// Mitsubishi GX Works2 project: pneumatic_control_3   PLC: Q03UDV

PROGRAM MAIN
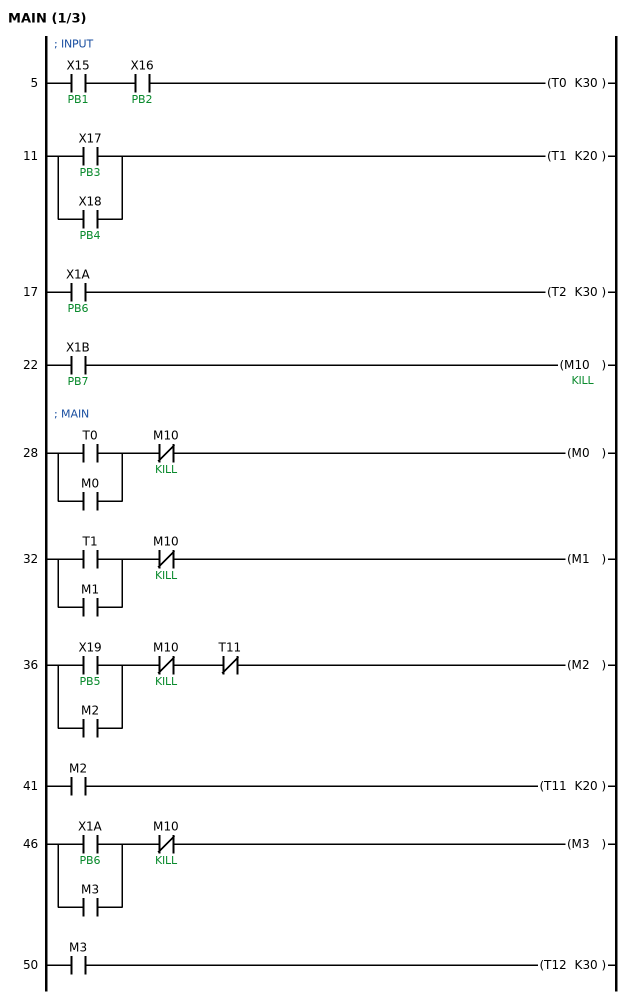
; INPUT
5     LD      X15  ; PB1
      AND     X16  ; PB2
      OUT     T0 K30
11    LD      X17  ; PB3
      OR      X18  ; PB4
      OUT     T1 K20
17    LD      X1A  ; PB6
      OUT     T2 K30
22    LD      X1B  ; PB7
      OUT     M10  ; KILL
; MAIN
28    LD      T0
      OR      M0
      ANI     M10  ; KILL
      OUT     M0
32    LD      T1
      OR      M1
      ANI     M10  ; KILL
      OUT     M1
36    LD      X19  ; PB5
      OR      M2
      ANI     M10  ; KILL
      ANI     T11
      OUT     M2
41    LD      M2
      OUT     T11 K20
46    LD      X1A  ; PB6
      OR      M3
      ANI     M10  ; KILL
      OUT     M3
50    LD      M3
      OUT     T12 K30
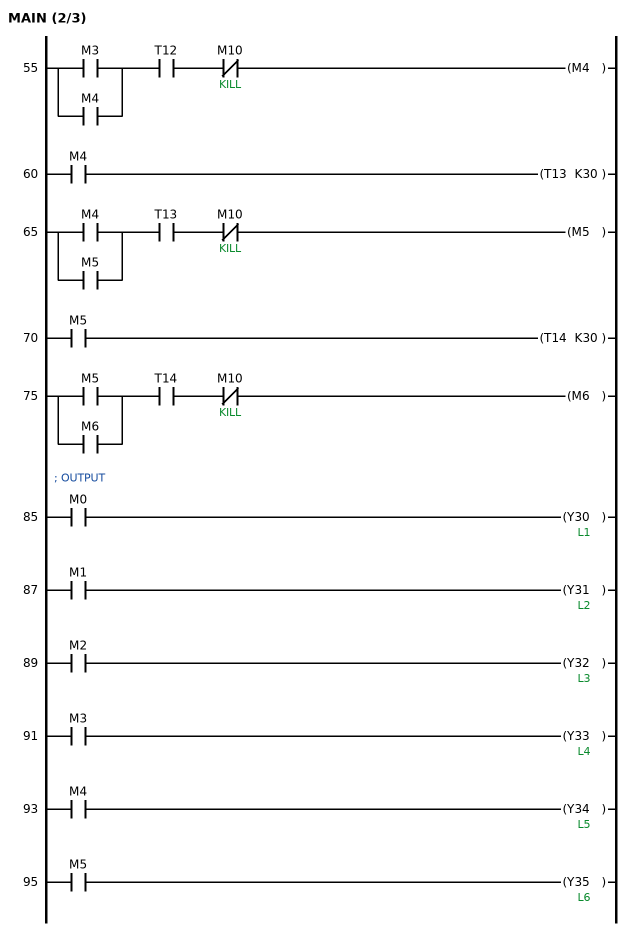
55    LD      M3
      OR      M4
      AND     T12
      ANI     M10  ; KILL
      OUT     M4
60    LD      M4
      OUT     T13 K30
65    LD      M4
      OR      M5
      AND     T13
      ANI     M10  ; KILL
      OUT     M5
70    LD      M5
      OUT     T14 K30
75    LD      M5
      OR      M6
      AND     T14
      ANI     M10  ; KILL
      OUT     M6
; OUTPUT
85    LD      M0
      OUT     Y30  ; L1
87    LD      M1
      OUT     Y31  ; L2
89    LD      M2
      OUT     Y32  ; L3
91    LD      M3
      OUT     Y33  ; L4
93    LD      M4
      OUT     Y34  ; L5
95    LD      M5
      OUT     Y35  ; L6
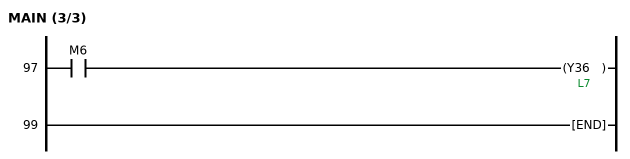
97    LD      M6
      OUT     Y36  ; L7
99    END
END_PROGRAM

// device comments not shown above
X1  ; RS1-1
X2  ; RS1-2
X3  ; RS2-1
X4  ; RS2-2
X1C  ; X1B
Y38  ; S/V1-1
Y39  ; S/V1-2
Y3A  ; S/V2
